{attribute 'GeneratedUsingTerminal: EP3204-0002-0017'}
{attribute addProperty BoxType "EP3204-0002-0017"}
{attribute addProperty Id "EtcSlaveTerminalBaseRTD_RTDInputs_Channel_1AT %I*RTD_RTDInputs_Channel_A8DF64E310RTD_RTDInputs_Channel_2AT %I*RTD_RTDInputs_Channel_A8DF64E310RTD_RTDInputs_Channel_3AT %I*RTD_RTDInputs_Channel_A8DF64E310RTD_RTDInputs_Channel_4AT %I*RTD_RTDInputs_Channel_A8DF64E310WcStateAT %I*WcState_9091E0EB2InfoDataAT %I*InfoData_32EB74EA10"}
{attribute addProperty CRC "2046876958"}
{attribute addProperty Size "52"}
TYPE EP3204_7A00DD1E EXTENDS EtcSlaveTerminalBase :
STRUCT
	{attribute addProperty Name "RTD_RTDInputs_Channel_1"}
	RTD_RTDInputs_Channel_1 : RTD_RTDInputs_Channel_A8DF64E3;
	{attribute addProperty Name "RTD_RTDInputs_Channel_2"}
	RTD_RTDInputs_Channel_2 : RTD_RTDInputs_Channel_A8DF64E3;
	{attribute addProperty Name "RTD_RTDInputs_Channel_3"}
	RTD_RTDInputs_Channel_3 : RTD_RTDInputs_Channel_A8DF64E3;
	{attribute addProperty Name "RTD_RTDInputs_Channel_4"}
	RTD_RTDInputs_Channel_4 : RTD_RTDInputs_Channel_A8DF64E3;
	{attribute addProperty Name "WcState"}
	WcState : WcState_9091E0EB;
	{attribute addProperty Name "InfoData"}
	InfoData : InfoData_32EB74EA;
END_STRUCT
END_TYPE

(* stored: Version 1.2.0.0, ProductVersion 3.1.4024.9
   DUT EP3204_7A00DD1E: Id {a5ab4274-9cd8-450d-8f6c-121a10012810} *)
